FUNCTION_BLOCK FB_Waage
	VAR_IN_OUT
		bNullsetzen	: BOOL;
	END_VAR
	
	VAR_OUTPUT
		iMesswert : INT;
	END_VAR
	
	VAR
		busyRec : BOOL;
		recError : ComError_t;
		bGotString : BOOL;
		
		arbeitsString : STRING;
		stringLange : INT;
	END_VAR
	
	
// ----- Ende der Definition. Hier folgt der Code ------

	// Nullsetzten der Waage
	IF bNullsetzen THEN
		bNullsetzen:= FALSE;
		TxWaage(SendString:= '<t>', Busy=> , Error=> , TXbuffer:= TxBufferWaage);
	END_IF
	
	
	
	
	// Messwert erhalten
	RecWaage(
		Prefix:= 'N  ', 
		Suffix:= ' g', 
		StringReceived=> bGotString, 
		Busy=> busyRec, 
		Error=> recError, 
		ReceivedString:= IFC_HW.waageNachricht, 
		RXbuffer:= RxBufferWaage);
	
	// Messwert als INT extrahieren
	arbeitsString := DELETE(STR:= IFC_HW.waageNachricht, POS:=1, LEN:=1);		// Beginn loschen
	stringLange := LEN(STR:=arbeitsString);
	arbeitsString := DELETE(STR:=arbeitsString, POS:= stringLange-1, LEN:=2);	// Ende loschen
	iMesswert := STRING_TO_INT(arbeitsString);									// String to int

END_FUNCTION_BLOCK

(* stored: Version 1.1.0.1, ProductVersion 3.1.4024.6
   POU FB_Waage: Id {074c83d0-e1d0-4825-bd99-e89e26c0b2cd}, SpecialFunc None *)
